TYPE tempData : 
STRUCT
	temp: REAL;
END_STRUCT
END_TYPE

(* stored: Version 1.1.0.1, ProductVersion 3.1.4024.12
   DUT tempData: Id {13f78209-136c-4be7-a05f-e21ea4d3dcc4} *)
